FUNCTION_BLOCK CMP_OC_W1

VAR_INPUT
	BOOL_INTERLOCK : BOOL; (*INTERLOCK*)
	WORD_1: WORD;		(*WORD 1*)
	END_VAR


VAR_OUTPUT
	BZ_OUTPUT_BOOL : BOOL;
END_VAR


VAR
	OUT_1: BOOL;
END_VAR

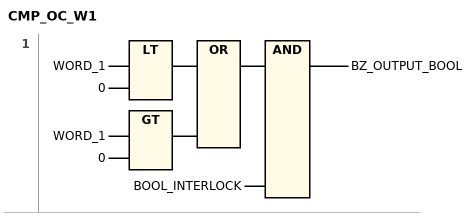
// NETWORK 1
BZ_OUTPUT_BOOL := (WORD_1 < 0 OR WORD_1 > 0) AND BOOL_INTERLOCK;

END_FUNCTION_BLOCK

(* stored: Version 1.1.0.1, ProductVersion 3.1.4024.12
   POU CMP_OC_W1: Id {e0046c2b-d0aa-4035-8b75-cff26dc2353c}, SpecialFunc None *)
